// TIA Portal V19 export
DATA_BLOCK "DB_ToHmi"   // DB28
{ S7_Optimized_Access := 'TRUE'; DB_Accessible_From_OPC_UA := 'FALSE' }
// stored: AutoNumber false, DBAccessibleFromOPCUA false, DBAccessibleFromWebserver false, MemoryReserve 100
   VAR
      xShowPopReqChangeBigbag : Bool;   // Show Popup change Bigbag requested
      xShowPopNoMoreRecipeAvailable : Bool;   // Show Popup no more recipe available in the data base
      xSafetyState { ExternalWritable := 'False'} : Bool;   // Safety State
      xDiseableRecipeButton { ExternalWritable := 'False'} : Bool;   // Diseable all button for manage recipe
      xDisplayPrevButton { ExternalWritable := 'False'} : Bool;   // Display previous button in recipe screen
      xDisplayNextButton { ExternalWritable := 'False'} : Bool;   // Display next button in recipe screen
      xDiseableNewButton { ExternalWritable := 'False'} : Bool;   // Diseable new recipe button
      xDiseableSaveButton { ExternalWritable := 'False'} : Bool;   // Diseable save recipe button
      xDiseableDeleteButton { ExternalWritable := 'False'} : Bool;   // Diseable delete recipe button
      xLockRecipe { ExternalWritable := 'False'} : Bool;   // Lock recipe during production
      xLockSelectJobDataNumber { ExternalWritable := 'False'} : Bool;   // Lock selection of job data number
      xLockJobDataLeft { ExternalWritable := 'False'} : Bool;   // Lock modification Job Data left robot
      xLockJobDataRight { ExternalWritable := 'False'} : Bool;   // Lock modification Job Data right robot
      xVacuumPumpRunning { ExternalWritable := 'False'} : Bool;
      xVacuumDriveActivated { ExternalWritable := 'False'} : Bool;
      xLockMaintenance { ExternalWritable := 'False'} : Bool;   // Lock button to switch in Maintenance mode
      xLockSemiAuto { ExternalWritable := 'False'} : Bool;   // Lock button to switch in Semi-Auto mode
      xHomePositionR1 { ExternalWritable := 'False'} : Bool;   // Robot 1 in Home Position
      xHomePositionR2 { ExternalWritable := 'False'} : Bool;   // Robot 2 in Home Position
      xAccessDoor { ExternalWritable := 'False'} : Bool;   // Access door closed
      xCaptiveKey { ExternalWritable := 'False'} : Bool;   // Captive key on contact switch
      xLightBeam { ExternalWritable := 'False'} : Bool;   // Light Beam clear
      xCbsGate { ExternalWritable := 'False'} : Bool;   // CBS Gate closed
      nGlobalState { ExternalWritable := 'False'} : Int;   // Cell global state
      wVacuumState { ExternalWritable := 'False'} : Word;
      uiProdRecordMin { ExternalWritable := 'False'} : UInt;   // Mini record number
      uiProdRecordMax { ExternalWritable := 'False'} : UInt;   // Maxi record number
      uiFlatRecMinLeftRobot { ExternalWritable := 'False'} : UInt;   // Mini record number for Flatness Left robot
      uiFlatRecMaxLeftRobot { ExternalWritable := 'False'} : UInt;   // Maxi record number for Flatness Left robot
      uiFlatRecMinRightRobot { ExternalWritable := 'False'} : UInt;   // Mini record number for Flatness Right robot
      uiFlatRecMaxRightRobot { ExternalWritable := 'False'} : UInt;   // Maxi record number for Flatness Right robot
      uiNbrDisplyedLine { ExternalWritable := 'False'} : UInt;   // Number of displayed lime of production
      uiFirstRecordDisplayed { ExternalWritable := 'False'} : UInt;   // First record displayed
      uiLastRecordDisplayed { ExternalWritable := 'False'} : UInt;   // Last record displayed
      sVacuumRunningTime { ExternalWritable := 'False'} : String[15];
      LeftRobot : Struct
         xRobotInAuto { ExternalWritable := 'False'} : Bool;
         xRobotInManu { ExternalWritable := 'False'} : Bool;
         xRobotReqReset { ExternalWritable := 'False'} : Bool;
         xRecipeInProgress { ExternalWritable := 'False'} : Bool;
         xPathInProgress { ExternalWritable := 'False'} : Bool;   // Service path in progress
         xPathStopped { ExternalWritable := 'False'} : Bool;   // Service path stopped
         xPathCancelled { ExternalWritable := 'False'} : Bool;   // Service path cancelled
         xContactState { ExternalWritable := 'False'} : Bool;   // State of the FerRobotic head contact
         xShowPopRemoveDisk : Bool;
         xShowPopPickupDisk : Bool;
         xShowPopFlatnessFault : Bool;
         xMagazineEmpty { ExternalWritable := 'False'} : Bool;
         xRangeFinderDetection { ExternalWritable := 'False'} : Bool;
         xValveOpen { ExternalWritable := 'False'} : Bool;
         xValveClosed { ExternalWritable := 'False'} : Bool;
         uiRangeFinderValue { ExternalWritable := 'False'} : UInt;
         nActualForce { ExternalWritable := 'False'} : Int;   // Actual force on FerRobotic head
         rActualPosition { ExternalWritable := 'False'} : Real;   // Actual position of the FerRobotic head
         uiActualJobDataNumber { ExternalWritable := 'False'} : UInt;
         uiNbDiskUsed { ExternalWritable := 'False'} : UInt;
         uiRobotStatus { ExternalWritable := 'False'} : UInt;
         uiSetSpeed { ExternalWritable := 'False'} : UInt;
         uiRobotSpeed { ExternalWritable := 'False'} : UInt;
         uiPaperChangeDistance { ExternalWritable := 'False'} : UInt;
         uiCounterPulse_X { ExternalWritable := 'False'} : UInt;
         uiCounterPulse_Z { ExternalWritable := 'False'} : UInt;
         uiGreaseFault_X { ExternalWritable := 'False'} : UInt;
         uiGreaseFault_Z { ExternalWritable := 'False'} : UInt;
         uiDistanceSandingDisk { ExternalWritable := 'False'} : UInt;
         uiActualRobotSpeed { ExternalWritable := 'False'} : UInt;   // Actual speed of theTCP of the robot
         uiDistanceBeforeGreasingX : UInt;
         uiDistanceBeforeGreasingZ : UInt;
         udiOdometer_X { ExternalWritable := 'False'} : UDInt;
         udiOdometer_Z { ExternalWritable := 'False'} : UDInt;
         sRunTime { ExternalWritable := 'False'} : String[12];
         sPauseTime { ExternalWritable := 'False'} : String[12];
         sFaultTime { ExternalWritable := 'False'} : String[12];
         sRobotPowerOnTime { ExternalWritable := 'False'} : String[15];
         sRobotDriveOnTime { ExternalWritable := 'False'} : String[15];
         IB_Safety500 { ExternalWritable := 'False'} : SInt;
         IB_Input100 { ExternalWritable := 'False'} : SInt;
         IB_Input101 { ExternalWritable := 'False'} : SInt;
         IB_Input102 { ExternalWritable := 'False'} : SInt;
         IB_Input103 { ExternalWritable := 'False'} : SInt;
         IN_Input600 { ExternalWritable := 'False'} : Int;
         IN_Input602 { ExternalWritable := 'False'} : Int;
         IN_Input604 { ExternalWritable := 'False'} : Int;
         IN_Input606 { ExternalWritable := 'False'} : Int;
         OB_Safety508 { ExternalWritable := 'False'} : SInt;
         OB_Output100 { ExternalWritable := 'False'} : SInt;
         OB_Output101 { ExternalWritable := 'False'} : SInt;
         IB_Fast90 { ExternalWritable := 'False'} : SInt;
      END_STRUCT;
      RightRobot : Struct
         xRobotInAuto { ExternalWritable := 'False'} : Bool;
         xRobotInManu { ExternalWritable := 'False'} : Bool;
         xRobotReqReset { ExternalWritable := 'False'} : Bool;
         xRecipeInProgress { ExternalWritable := 'False'} : Bool;
         xPathInProgress { ExternalWritable := 'False'} : Bool;   // Service path in progress
         xPathStopped { ExternalWritable := 'False'} : Bool;   // Service path stopped
         xPathCancelled { ExternalWritable := 'False'} : Bool;   // Service path cancelled
         xContactState { ExternalWritable := 'False'} : Bool;   // State of the FerRobotic head contact
         xShowPopRemoveDisk : Bool;
         xShowPopPickupDisk : Bool;
         xShowPopFlatnessFault : Bool;
         xMagazineEmpty { ExternalWritable := 'False'} : Bool;
         xRangeFinderDetection { ExternalWritable := 'False'} : Bool;
         xValveOpen { ExternalWritable := 'False'} : Bool;
         xValveClosed { ExternalWritable := 'False'} : Bool;
         uiRangeFinderValue { ExternalWritable := 'False'} : UInt;
         nActualForce { ExternalWritable := 'False'} : Int;   // Actual force on FerRobotic head
         rActualPosition { ExternalWritable := 'False'} : Real;   // Actual position of the FerRobotic head
         uiActualJobDataNumber { ExternalWritable := 'False'} : UInt;
         uiNbDiskUsed { ExternalWritable := 'False'} : UInt;
         uiRobotStatus { ExternalWritable := 'False'} : UInt;
         uiSetSpeed { ExternalWritable := 'False'} : UInt;
         uiRobotSpeed { ExternalWritable := 'False'} : UInt;
         uiPaperChangeDistance { ExternalWritable := 'False'} : UInt;
         uiCounterPulse_X { ExternalWritable := 'False'} : UInt;
         uiCounterPulse_Z { ExternalWritable := 'False'} : UInt;
         uiGreaseFault_X { ExternalWritable := 'False'} : UInt;
         uiGreaseFault_Z { ExternalWritable := 'False'} : UInt;
         uiDistanceSandingDisk { ExternalWritable := 'False'} : UInt;
         uiActualRobotSpeed { ExternalWritable := 'False'} : UInt;   // Actual speed of theTCP of the robot
         uiDistanceBeforeGreasingX : UInt;
         uiDistanceBeforeGreasingZ : UInt;
         udiOdometer_X { ExternalWritable := 'False'} : UDInt;
         udiOdometer_Z { ExternalWritable := 'False'} : UDInt;
         sRunTime { ExternalWritable := 'False'} : String[12];
         sPauseTime { ExternalWritable := 'False'} : String[12];
         sFaultTime { ExternalWritable := 'False'} : String[12];
         sRobotPowerOnTime { ExternalWritable := 'False'} : String[15];
         sRobotDriveOnTime { ExternalWritable := 'False'} : String[15];
         IB_Safety500 { ExternalWritable := 'False'} : SInt;
         IB_Input100 { ExternalWritable := 'False'} : SInt;
         IB_Input101 { ExternalWritable := 'False'} : SInt;
         IB_Input102 { ExternalWritable := 'False'} : SInt;
         IB_Input103 { ExternalWritable := 'False'} : SInt;
         IN_Input600 { ExternalWritable := 'False'} : Int;
         IN_Input602 { ExternalWritable := 'False'} : Int;
         IN_Input604 { ExternalWritable := 'False'} : Int;
         IN_Input606 { ExternalWritable := 'False'} : Int;
         OB_Safety508 { ExternalWritable := 'False'} : SInt;
         OB_Output100 { ExternalWritable := 'False'} : SInt;
         OB_Output101 { ExternalWritable := 'False'} : SInt;
         IB_Fast90 { ExternalWritable := 'False'} : SInt;
      END_STRUCT;
      aRecipeList { ExternalWritable := 'False'} : Array[1..10] of "stRecipeListHMI";   // List of the recipe name display on HMI
      DataSentronMainPanel { ExternalWritable := 'False'} : "Sentron_PAC";   // Sentron main panel data
      DateSentronLeftRobot { ExternalWritable := 'False'} : "Sentron_PAC";   // Sentron left robot data
      DataSentronRightRobot { ExternalWritable := 'False'} : "Sentron_PAC";   // Sentron right robot data
      Fault { ExternalWritable := 'False'} : Struct
         wFerRoboticLeft : Word;
         wManageRobotLeft : Word;
         wOtherLeft : Word;
         wRobotLeft : Word;
         wVacuumValveLeft : Word;
         wFerRoboticManageLeft : Word;
         wFault07 : Word;
         wFault08 : Word;
         wFerRoboticRight : Word;
         wManageRobotRight : Word;
         wOtherRight : Word;
         wRobotRight : Word;
         wVacuumValveRight : Word;
         wFerRoboticManageRight : Word;
         wFault11 : Word;
         wFault12 : Word;
         wSafetFault : Word;
         wVacuumFault : Word;
         wSafetyModule : Word;
         wOtherMaster : Word;
         wFault15 : Word;
         wFault16 : Word;
         wFault17 : Word;
         wFault18 : Word;
      END_STRUCT;
      Warning { ExternalWritable := 'False'} : Struct
         wSafetyComp : Word;
         wWarnigLeft : Word;
         wWarnigRight : Word;
         wWarnig04 : Word;
         wWarnig05 : Word;
         wWarnig06 : Word;
         wWarnig07 : Word;
         wWarnig08 : Word;
         wWarnig09 : Word;
         wWarnig10 : Word;
      END_STRUCT;
      Message { ExternalWritable := 'False'} : Struct
         wMessage01 : Word;
         wMessage02 : Word;
         wMessage03 : Word;
         wMessage04 : Word;
      END_STRUCT;
      aDisplayProdData { ExternalWritable := 'False'} : Array[0..9] of "stProductionRecord";
      DisplayFlatRecLeftRobot { ExternalWritable := 'False'} : "stFlatnessCtrlRecord";
      DisplayFlatRecRightRobot { ExternalWritable := 'False'} : "stFlatnessCtrlRecord";
   END_VAR
BEGIN
END_DATA_BLOCK
